FUNCTION_BLOCK ABSTRACT FB_StopperVetoable
VAR
    {attribute 'pytmc' := '
        pv: StopperMask
        io: i
        field: DESC Bitmask of stoppers that veto this
    '}
    wStopperMask : WORD;
    fbLog : FB_LogMessage;
END_VAR

METHOD AddStopper : BOOL
VAR_INPUT
    wStopper: WORD;
END_VAR
AddStopper := WORD_TO_BOOL(wStopperMask AND SHL(WORD#1, wStopper));
wStopperMask := wStopperMask OR SHL(WORD#1, wStopper);
END_METHOD

METHOD CheckStoppers : BOOL
VAR
    i: WORD;

    StopperPairing : ARRAY[1..PMPS_GVL.MAX_VETO_DEVICES] OF WORD;
END_VAR
CheckStoppers := FALSE;
{IF defined (K)}
    StopperPairing := PMPS_GVL.K_Stopper_Pairings;
{ELSIF defined (L)}
    StopperPairing := PMPS_GVL.L_Stopper_Pairings;
{ELSE}
    fbLog(sMsg := 'K/L compiler definition missing.', eSevr := TcEventSeverity.Critical);
    RETURN;
{END_IF}

FOR i:=1 TO (PMPS_GVL.MAX_VETO_DEVICES-1) BY 1 DO
    IF PMPS_GVL.stCurrentBeamParameters.aVetoDevices[i] AND WORD_TO_BOOL(wStopperMask AND SHL(WORD#1, i)) THEN
        IF StopperPairing[i] <> 0 AND StopperPairing[i] <> PMPS_GVL.MAX_VETO_DEVICES THEN
            IF NOT PMPS_GVL.stCurrentBeamParameters.aVetoDevices[StopperPairing[i]] AND NOT WORD_TO_BOOL(wStopperMask AND SHL(WORD#1, StopperPairing[i])) THEN
                CheckStoppers := TRUE;
                RETURN;
            END_IF
        ELSE
            CheckStoppers := TRUE;
            RETURN;
        END_IF
    END_IF
END_FOR
END_METHOD

METHOD RemoveStopper : BOOL
VAR_INPUT
    wStopper: WORD;
END_VAR
RemoveStopper := WORD_TO_BOOL(wStopperMask AND SHL(WORD#1, wStopper));
wStopperMask := wStopperMask AND NOT SHL(WORD#1, wStopper);
END_METHOD

END_FUNCTION_BLOCK

(* stored: Version 1.1.0.1, ProductVersion 3.1.4026.12
   POU FB_StopperVetoable: Id {9114ce33-096d-4859-8327-51a29b1b7c16}, SpecialFunc None
   Method AddStopper: Id {dfc9400d-efbb-4f3c-bb34-86649ddea037}
   Method CheckStoppers: Id {1e391055-0614-47cf-92fe-50cbf0483ad1}
   Method RemoveStopper: Id {00072576-a6e6-4097-9bd8-6246e1ae5421} *)
